FUNCTION F_GetTwoLineAngle : LREAL	//ermittelt den Winkel zwischen zwei Linien in XY-Ebene
VAR_INPUT
	line1_P1 : ST_3DPoint;
	line1_P2 : ST_3DPoint;
	line2_P1 : ST_3DPoint;
	line2_P2 : ST_3DPoint;	
END_VAR
VAR
	vec1X, vec1Y, vec2X, vec2Y : LREAL;
	temp : LREAL;
	angle1 : LREAL;
	angle2 : LREAL;
END_VAR

//1. Linien in Ortsvektoren umrechnen
vec1X := line1_P2.X - line1_P1.X;
vec1Y := line1_P2.Y - line1_P1.Y;

vec2X := line2_P2.X - line2_P1.X;
vec2Y := line2_P2.Y - line2_P1.Y;

//Vektor 1 auf Einheitskreis normalisieren
//Länge berechnen
temp := vec1X * vec1X + vec1Y * vec1Y;
IF temp = 0.0 THEN
	F_GetTwoLineAngle := 9999.9; //führt zu Wurzel aus "0" was bedeutet, dass der Vektor keine Länge hat
	RETURN;
END_IF
temp := SQRT(temp);
//normalisieren 
vec1X := vec1X / temp;
vec1Y := vec1Y / temp;

//Vektor 2 auf Einheitskreis normalisieren
//Länge berechnen
temp := vec2X * vec2X + vec2Y * vec2Y;
IF temp = 0.0 THEN
	F_GetTwoLineAngle := 9999.9; //führt zu Wurzel aus "0" was bedeutet, dass der Vektor keine Länge hat
	RETURN;
END_IF
temp := SQRT(temp);
//normalisieren 
vec2X := vec2X / temp;
vec2Y := vec2Y / temp;

//Winkelberechnung Vektor 1 in Bezug zu X-Achse im Koordinatensystem
IF vec1Y < 0.0 THEN	//Vektor befindet sich im Quadranten III oder IV
	angle1 := 360.0 -  RAD_TO_DEG(ACOS(vec1X));
ELSE
	angle1 := RAD_TO_DEG(ACOS(vec1X));
END_IF

//Winkelberechnung Vektor 2 in Bezug zu X-Achse im Koordinatensystem
IF vec2Y < 0.0 THEN	//Vektor befindet sich im Quadranten III oder IV
	angle2 := 360.0 -  RAD_TO_DEG(ACOS(vec2X));
ELSE
	angle2 := RAD_TO_DEG(ACOS(vec2X));
END_IF

F_GetTwoLineAngle := angle2 - angle1;

IF F_GetTwoLineAngle > 180.0 THEN
	F_GetTwoLineAngle := F_GetTwoLineAngle - 360.0;
END_IF

END_FUNCTION

(* stored: Version 1.1.0.1, ProductVersion 3.1.4020.12
   POU F_GetTwoLineAngle: Id {f5f92eff-cb2a-47b4-94bf-e297b649390c}, SpecialFunc None *)
